FUNCTION_BLOCK TankCtrl_Disabled EXTENDS _TankCtrl_State

METHOD OnExecute
IF _ctx.hmi.bMultiButton THEN
	_ctx.hmi.bMultiButton := FALSE;
	
	_ctx.priv.smgr.Request(_ctx.state.iEnabled);
END_IF
END_METHOD

METHOD OnInit
_ctx.hmi.bMultiButtonVis := TRUE;
_ctx.hmi.nMultiButtonColor := COL.ORANGE.Raw;
_ctx.hmi.nMultiButtonText := 'Press to  Enable';

_ctx.priv.IsSystemOn.Lower();

_ctx.io.out.bRunPump := FALSE;
END_METHOD

END_FUNCTION_BLOCK

(* stored: Version 1.1.0.1
   POU TankCtrl_Disabled: Id {427c8205-4cc9-476e-88c9-78dfc63362ce}, SpecialFunc None
   Method OnExecute: Id {0ffa6e9a-cfe8-4551-a6fc-51c65774b1c6}
   Method OnInit: Id {6c85ef7e-9de4-410f-979e-f08a56ae0eb6} *)
